PROGRAM P_Lys_Grp0
VAR
	fbLight_GRP0: FB_DALILgtActr_EX;
	eMod: SH_Light.E_DALIAddressType := SH_Light.E_DALIAddressType.Group;
	fSttupCtrlVal: REAL;
	fMinCtrlVal: REAL := 0;
	fMaxCtrlVal: REAL := 100;
	fLgtOffset: REAL := 5;
	eFadeTime: SH_Light.E_DALIFadeTime := SH_Light.E_DALIFadeTime.T02000ms;
	eFadeRate: SH_Light.E_DALIFadeRate := SH_Light.E_DALIFadeRate.N063StepsPerSec;
	uiBlinkTi: UINT := 2;
	uiOffDly: UINT := 0;
	uiPollActLgtLvl: UINT := 30;
	bReInit: BOOL;
	nCycleTimeInMS: UDINT := 10;
	stLgtCmd: SH_Light.ST_LgtCmd;
END_VAR

VAR CONSTANT
	DALI_LINE_NUM: BYTE := 1;
END_VAR

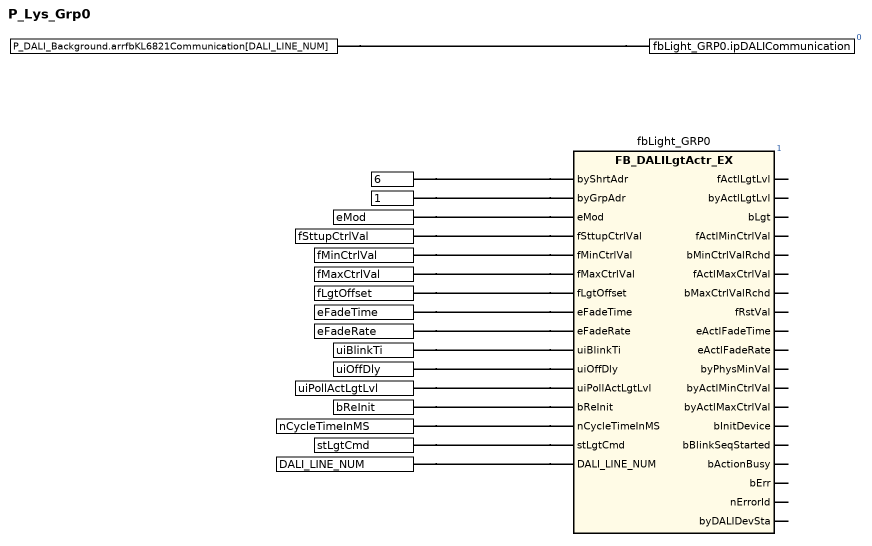
fbLight_GRP0.ipDALICommunication := P_DALI_Background.arrfbKL6821Communication[DALI_LINE_NUM];
fbLight_GRP0(
    byShrtAdr := 6,
    byGrpAdr := 1,
    eMod := eMod,
    fSttupCtrlVal := fSttupCtrlVal,
    fMinCtrlVal := fMinCtrlVal,
    fMaxCtrlVal := fMaxCtrlVal,
    fLgtOffset := fLgtOffset,
    eFadeTime := eFadeTime,
    eFadeRate := eFadeRate,
    uiBlinkTi := uiBlinkTi,
    uiOffDly := uiOffDly,
    uiPollActLgtLvl := uiPollActLgtLvl,
    bReInit := bReInit,
    nCycleTimeInMS := nCycleTimeInMS,
    stLgtCmd := stLgtCmd,
    DALI_LINE_NUM := DALI_LINE_NUM); // FB_DALILgtActr_EX

END_PROGRAM

(* stored: Version 1.1.0.1
   POU P_Lys_Grp0: Id {6f72ea74-fce5-4ebf-a2a8-56b8ba1812ea}, SpecialFunc None *)
